KUKA KRL program: makrosps2.src

&ACCESS RV
&PARAM TEMPLATE = C:\KRC\Roboter\Template\makrospsvorgabe.src
&PARAM EDITMASK = MakroSPS2
&PARAM TPVW_VERSION=8.3.18
DEF MAKROSPS2 ( )
; FOLD Makro Anfang;%{PSE} %MKUKATPVW
SPS_N=-1
; ENDFOLD
; FOLD ;%{H}
END
; ENDFOLD
